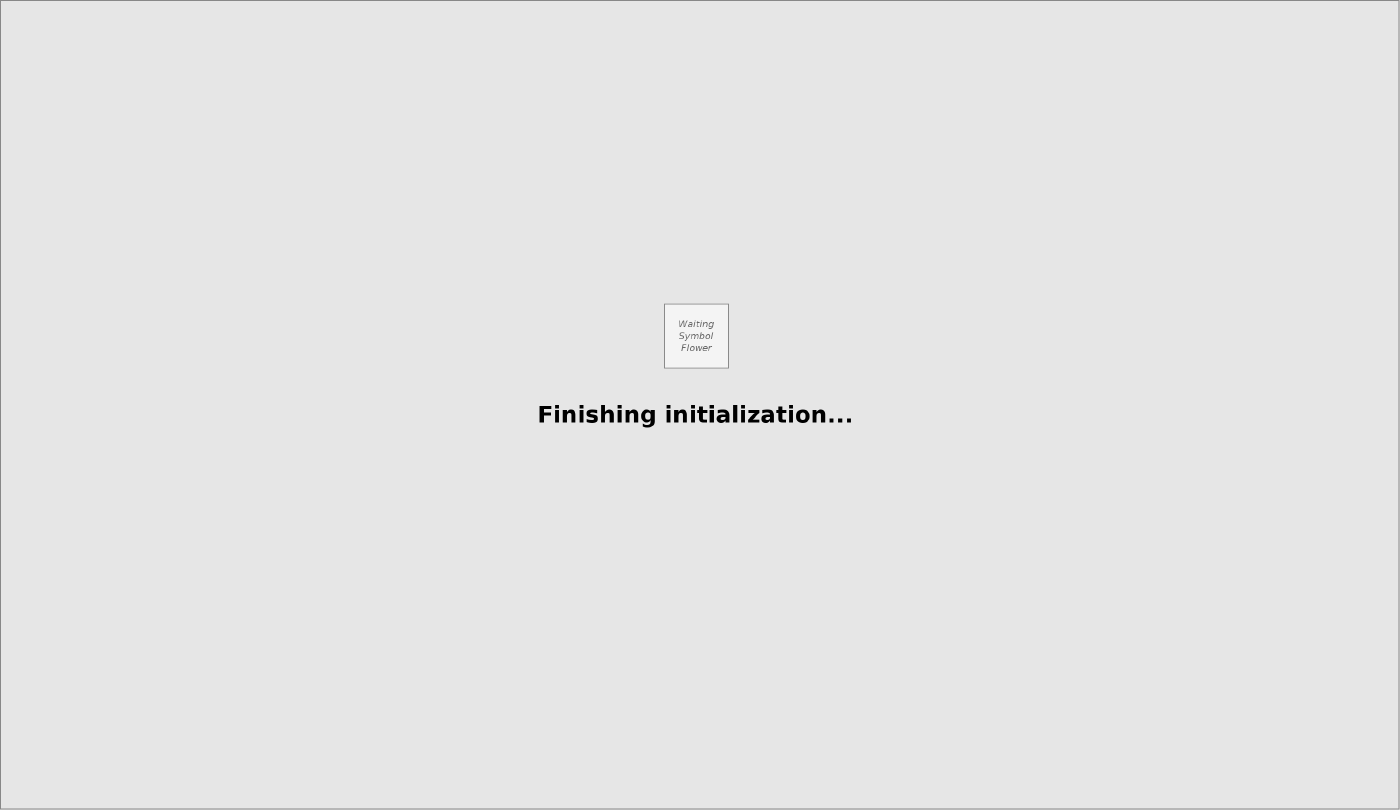
VISUALIZATION PageReadyInitialized_1  // 1520x880
    WaitingSymbolFlower (721,330 70x70)
    Label (530,430 450x40), "Finishing initialization..."
END_VISUALIZATION

(* stored: Version 1.1.0.1, ProductVersion 3.1.4024.12
   Visu PageReadyInitialized_1: Id {46acdf14-4801-41dc-9def-a3020f8f9361} *)
